// TIA Portal V19 export
VAR_GLOBAL   // PLC tag table "Digital"
END_VAR
